# B&R Automation Studio project Lab1_RMS
Automation Studio 4.5.2.102

## Configuration Config1

### Task classes (Cpu.sw)
```
Cyclic#4 (cycle 20000 us, tolerance 20000 us):
  Program <- Program.prg
Libraries: MotorContr
```

### Hardware
```
4PP065_0571_P74 : 4PP065.0571-P74 v1.1.2.0
  Connector IF5:
    ActivateDevice = 1
    Mode = Manual
    InternetAddress = 10.0.1.11
    SubnetMask = 255.255.255.0
  ConfigurationID = labBR
  Cyclic4Duration = 20000
  Cyclic4Tolerance = 20000
```

## Logical view

### Global.var - Global variables
```iecst
VAR
	btn1 : BOOL;
END_VAR
```

### Library Logical/MotorContr (ANSIC)

#### MotorContr.fun - Exported functions and function blocks
```iecst
{REDUND_ERROR} FUNCTION_BLOCK FB_motor (*FB motorrrrrrrrrrrrrrrrrrrrrrrrr*) (*$GROUP=User,$CAT=User,$GROUPICON=User.png,$CATICON=User.png*)
	VAR_INPUT
		u : {REDUND_UNREPLICABLE} REAL;
	END_VAR
	VAR_OUTPUT
		w : {REDUND_UNREPLICABLE} REAL;
		phi : {REDUND_UNREPLICABLE} REAL;
	END_VAR
	VAR
		w_integrator : {REDUND_UNREPLICABLE} FB_Integrator;
		Tm : {REDUND_UNREPLICABLE} REAL;
		ke : {REDUND_UNREPLICABLE} REAL;
		dt : {REDUND_UNREPLICABLE} REAL;
		phi_integrator : FB_Integrator;
	END_VAR
END_FUNCTION_BLOCK

{REDUND_ERROR} {REDUND_UNREPLICABLE} FUNCTION_BLOCK FB_Integrator (*intrigal*) (*$GROUP=User,$CAT=User,$GROUPICON=User.png,$CATICON=User.png*)
	VAR_INPUT
		in : {REDUND_UNREPLICABLE} REAL;
	END_VAR
	VAR_OUTPUT
		out : {REDUND_UNREPLICABLE} REAL;
	END_VAR
	VAR
		dt : {REDUND_UNREPLICABLE} REAL;
		state : {REDUND_UNREPLICABLE} REAL;
	END_VAR
END_FUNCTION_BLOCK

{REDUND_ERROR} {REDUND_UNREPLICABLE} FUNCTION_BLOCK FB_regulator (*TODO: Add your comment here*) (*$GROUP=User,$CAT=User,$GROUPICON=User.png,$CATICON=User.png*)
	VAR_INPUT
		e : {REDUND_UNREPLICABLE} REAL;
	END_VAR
	VAR_OUTPUT
		u : {REDUND_UNREPLICABLE} REAL;
	END_VAR
	VAR
		k_p : {REDUND_UNREPLICABLE} REAL;
		k_i : {REDUND_UNREPLICABLE} REAL;
		integrator : {REDUND_UNREPLICABLE} FB_Integrator;
		iyOld : {REDUND_UNREPLICABLE} REAL;
		max_abs_value : {REDUND_UNREPLICABLE} REAL;
		dt : {REDUND_UNREPLICABLE} REAL;
	END_VAR
END_FUNCTION_BLOCK
```

#### FB_motor.c
```c
#include <bur/plctypes.h>
#ifdef __cplusplus
	extern "C"
	{
#endif
	#include "MotorContr.h"
#ifdef __cplusplus
	};
#endif

void FB_motor(struct FB_motor* inst)
{
	REAL bf1 = (inst->u) / inst->ke - inst->w;
	REAL bf2 = bf1 / inst->Tm;

	inst->w_integrator.in = bf2;
	FB_Integrator(&inst->w_integrator);
	inst->w = inst->w_integrator.out;

	inst->phi_integrator.in = inst->w;
	FB_Integrator(&inst->phi_integrator);
	inst->phi = inst->phi_integrator.out;
}
```

#### FB_Integrator.c
```c
#include <bur/plctypes.h>
#ifdef __cplusplus
	extern "C"
	{
#endif
	#include "MotorContr.h"
#ifdef __cplusplus
	};
#endif
/* intrigal */
void FB_Integrator(struct FB_Integrator* inst)
{
	inst->dt=0.002;
	inst->out = inst->dt * inst->in + inst->state;
	inst->state = inst->out;

}
```

#### FB_regulator.c
```c
#include <bur/plctypes.h>
#ifdef __cplusplus
	extern "C"
	{
#endif
	#include "MotorContr.h"
#ifdef __cplusplus
	};
#endif
/* TODO: Add your comment here */
void FB_regulator(struct FB_regulator* inst)
{
	REAL p_part = inst->e * inst->k_p;
	REAL i_part = inst->e * inst->k_i;

	inst->integrator.in = i_part;
	FB_Integrator(&inst->integrator);
	i_part = inst->integrator.out;

	REAL pi_reg = p_part + i_part;

	if (pi_reg > inst->max_abs_value) {
		inst->u = inst->max_abs_value;
		inst->integrator.out = inst->max_abs_value - p_part;
	} else if (pi_reg < -inst->max_abs_value) {
		inst->u = -inst->max_abs_value;
		inst->integrator.out = -inst->max_abs_value - p_part;
	} else {
		inst->u = pi_reg;
	}

	inst->iyOld = i_part;
}
```

### Program Logical/Program (ANSIC)

#### Variables.var
```iecst
VAR
	speed : REAL;
	enable : BOOL := TRUE;
	fb_regulator : FB_regulator;
	fb_motor : FB_motor;
	fb_motor2 : FB_motor;
	counter : INT;
END_VAR
```

#### Main.c
```c
#include <bur/plctypes.h>

#ifdef _DEFAULT_INCLUDES
	#include <AsDefault.h>
#endif

void _INIT ProgramInit(void)
{
	enable = 0;
	speed = 0;

	fb_regulator.dt = 0.002;
	fb_regulator.k_p = 0.45;
	fb_regulator.k_i = 10.0;
	fb_regulator.max_abs_value=24;

	fb_motor.dt = 0.002;
	fb_motor.ke = 4;
	fb_motor.Tm = 0.03;

	fb_motor2.dt = 0.002;
	fb_motor2.ke = 4;
	fb_motor2.Tm = 0.03;

}

void _CYCLIC ProgramCyclic(void)
{
	if (enable)
	{
		speed = 40.0;
	}
	else
	{
		speed = 0.0;
	}

	fb_regulator.e = speed - fb_motor.w;
	FB_regulator(&fb_regulator);

	fb_motor.u = 2*fb_regulator.u*fb_motor.ke;
	fb_motor2.u = speed*fb_motor2.ke;

	FB_motor(&fb_motor);
	FB_motor(&fb_motor2);
}

void _EXIT ProgramExit(void)
{

}
```

Listed in the project but not available here: Logical/Global.typ, Logical/Libraries, Logical/MotorContr/Types.typ, Logical/MotorContr/Constants.var
